// TIA Portal V21 export
TYPE "Tra_Motore_Formato"
TITLE = Motore1
   STRUCT
      Formati_Motore { S7_SetPoint := 'True'} : Array[0..10] of "Tra_Motore_dati";
   END_STRUCT;
END_TYPE
